{attribute 'qualified_only'}
{attribute 'strict'}
TYPE E_PulseState :
(
	SAFE			:= 0, //IDLE
	CHARGING		:= 1, //Charge
	CHARGECOMPLETE	:= 2, //EOC
	//DISCONNECTING	:= 3, //Disconnect
	DUMPING			:= 4, 
	//ABORT			:= 5,
	TRIPPED			:= 6	
);
END_TYPE

(* stored: Version 1.1.0.1, ProductVersion 3.1.4024.11
   DUT E_PulseState: Id {d8b04e17-a06a-475d-b7a6-e7e060a14014} *)
